// TIA Portal V17 export
// export: Created 2024-09-03T21:54:52.3990642Z, ExportSetting WithDefaults, DisplayName Totally Integrated Automation Portal, DisplayVersion V17 Update 7, DisplayName TIA Portal Openness, DisplayVersion V17 Update 7, DisplayName TIA Portal Version Control Interface, DisplayVersion V17, DisplayName SINAMICS Startdrive Advanced, DisplayVersion V17 SP2, DisplayName SINAMICS Startdrive G110M, G120, G120C, G120D, G120P, G115D, DisplayVersion V17 SP2, DisplayName SINAMICS Startdrive G130, G150, S120, S150, SINAMICS MV, S210, DisplayVersion V17 SP2, DisplayName STEP 7 Professional, DisplayVersion V17 Update 7, DisplayName STEP 7 Safety, DisplayVersion V17 Update 6, DisplayName WinCC Advanced / Unified PC, DisplayVersion V17 Update 7
DATA_BLOCK "Reader Parameters"   // DB300
{ S7_Optimized_Access := 'TRUE' }
VERSION : 0.1
// stored: AutoNumber false, DBAccessibleFromOPCUA true, DBAccessibleFromWebserver true, IsOnlyStoredInLoadMemory false, IsRetainMemResEnabled false, IsWriteProtectedInAS false, MemoryReserve 100
   VAR
      Reader : Array[1.."MaxReader"] of "UDT_CognexReaders";
   END_VAR
BEGIN
   Reader[1].HW.In.AcquisitionStatus := 424;
   Reader[1].HW.In.ResultsStatus := 422;
   Reader[1].HW.In.SoftEventControl := 388;
   Reader[1].HW.In.ResultData := 386;
   Reader[1].HW.Out.AcquisitionControl := 434;
   Reader[1].HW.Out.ResultsControl := 423;
   Reader[1].HW.Out.SoftEventControl := 388;
   Reader[1].HW.Out.UserData := 387;
END_DATA_BLOCK
